FUNCTION_BLOCK animacaoAbrirFechar (* Basic Function Block Type *)
  (* Standard: 61499-2 *)
  (* Version 0.0, 1/26/2026, Schneider Electric, Template *)
  PACKAGE Hidryco.HidrycoLib;
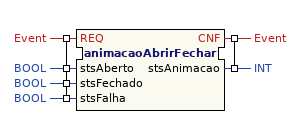
  EVENT_INPUT
    REQ WITH stsAberto, stsFechado, stsFalha; (* Normal Execution Request *)
  END_EVENT
  EVENT_OUTPUT
    CNF WITH stsAnimacao; (* Execution Confirmation *)
  END_EVENT
  VAR_INPUT
    stsAberto : BOOL;
    stsFechado : BOOL;
    stsFalha : BOOL;
  END_VAR
  VAR_OUTPUT
    stsAnimacao : INT; (* 0-Off; 1-On; 2-Fail; 3-Manut; 4-Transition *)
  END_VAR
  EC_STATES
    START; (* Initial State *)
    REQ;
  END_STATES
  ALGORITHM algREQ IN ST:
IF stsFalha THEN
    stsAnimacao := 2;       (* falha *)
ELSIF stsAberto AND stsFechado THEN
    stsAnimacao := 99;      (* fins de curso incoerentes: desconhecido *)
ELSIF stsAberto THEN
    stsAnimacao := 1;       (* aberto *)
ELSIF stsFechado THEN
    stsAnimacao := 0;       (* fechado *)
ELSE
    stsAnimacao := 4;       (* em trânsito *)
END_IF;
;
  END_ALGORITHM
END_FUNCTION_BLOCK
